FUNCTION_BLOCK I_PosDeltaHighPrecRapidUpd (* The "Position Delta, High Precision Rapid Update" Parameter Group is intended for applications where very high precision and very fast update rates are needed for position data. This PGN can provide delta position changes down to 1 millimeter with a delta time period accurate to 5 milliseconds *)
  (* Standard: NMEA 2000; Classification: PGN 129027; Function: Position Delta, High Precision Rapid Update; Description: Copyright (c) 2024 HR Agrartechnik GmbH This program and the accompanying materials are made available under the terms of the Eclipse Public License 2.0 which is available at https://www.eclipse.org/legal/epl-2.0/ SPDX-License-Identifier: EPL-2.0 https://docs.ms-muc-docs.de/projects/isobus-other-docs/de/latest/PGN/PGN_129026.html *)
  (* Version 1.0, 07.02.2025, Moritz Ortmeier, HR Agrartechnik GmbH *)
  PACKAGE isobus::tecu;
  (* Documentation:
  The "Position Delta, High Precision Rapid Update" Parameter Group is intended for applications where very high precision and very fast update rates are needed for position data. This PGN can provide delta position changes down to 1 millimeter with a delta time period accurate to 5 milliseconds
   TIMEOUT / IND Vertrag: TIMEOUT feuert ausschliesslich beim tatsaechlichen Eintreten eines Timeouts (Q_timeout wird true). Das Zuruecksetzen von Q_timeout auf false (Timeout vorbei) wird bewusst NICHT nochmal separat ueber TIMEOUT gemeldet, sondern kommt ueber IND - das feuert bei jedem Zyklus ohne aktiven Timeout und publiziert Q_timeout mit. Nachgeschaltete Bausteine, die auf das Ende eines Timeouts reagieren muessen, werten dafuer IND mit Q_timeout==false aus, nicht ein zweites TIMEOUT-Event.
  *)
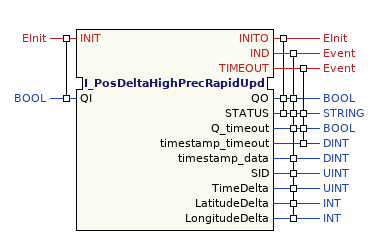
  EVENT_INPUT
    INIT : EInit WITH QI; (* Service Initialization *)
  END_EVENT
  EVENT_OUTPUT
    INITO : EInit WITH QO, STATUS; (* Initialization Confirm *)
    IND WITH QO, timestamp_data, SID, TimeDelta, LatitudeDelta, STATUS, Q_timeout, LongitudeDelta; (* Indication from Resource - feuert bei jedem Zyklus ohne aktiven Timeout und publiziert dabei auch den Reset von Q_timeout auf false. *)
    TIMEOUT WITH timestamp_timeout, STATUS, Q_timeout; (* Feuert ausschliesslich beim tatsaechlichen Eintreten eines Timeouts (Entry-Trigger). Das Zuruecksetzen von Q_timeout auf false wird NICHT hier, sondern ueber IND gemeldet. *)
  END_EVENT
  VAR_INPUT
    QI : BOOL; (* Event Input Qualifier *)
  END_VAR
  VAR_OUTPUT
    QO : BOOL; (* Event Output Qualifier *)
    STATUS : STRING;
    Q_timeout : BOOL;
    timestamp_timeout : DINT;
    timestamp_data : DINT;
    SID : UINT := UINT#16#FFFF; (* Sequence ID identifies the sequence this data is associated with so that the data can be synchronized with other vessel data for this same sequence being sent in another PGN. *)
    TimeDelta : UINT := UINT#16#FFFF;
    LatitudeDelta : INT := INT#16#7FFF;
    LongitudeDelta : INT := INT#16#7FFF;
  END_VAR
END_FUNCTION_BLOCK
